Fanuc KAREL source: kd00028.KL

-- PROVISIONAL review KL for V770-1; original PC SHA256 797bcf75f31c3fd704b93397fae550038d243d2089d9f1f0cdba8e347674be2a
-- Incomplete behavior may be omitted. Consult companion uncertainty JSON. Do not deploy.
PROGRAM KD00028
%NOLOCKGROUP
VAR
  I : INTEGER
  J : INTEGER
  B : BOOLEAN
  R : REAL
  S : STRING[80]
BEGIN
  -- UNRESOLVED_PC offsets 5-21; opcodes 9D,81,18,9D,12,22,9D,13,04
  -- UNRESOLVED_PC offsets 26-30; opcodes 7F
END KD00028
